FUNCTION_BLOCK DROP_SCREW
VAR_INPUT
END_VAR
VAR_OUTPUT
END_VAR
VAR
END_VAR

END_FUNCTION_BLOCK

(* stored: Version 1.1.0.1, ProductVersion 3.1.4022.18
   POU DROP_SCREW: Id {79fa5298-4375-4dd8-8def-d4665220c462}, SpecialFunc None *)
